# EPICS StreamDevice protocol: protocols/cpdac.proto
Terminator = LF;
ExtraInput = Ignore;
ReplyTimeout = 2500;

getMathSTA {
	out "math_\${1}_sta";
	in "%x";
}

clrMathSTA {
	out "math_\${1}_sta %x";
	in;
}

getProcSTA {
	out "proc_\${1}_sta";
	in "%x";
}

clrProcSTA {
	out "proc_\${1}_sta %x";
	in;
}

setBurstLen {
	out "burstlen %u";
	in;
}

setBurstMode {
	out "burstmode %u";
	in;
}
